(* IEC 61131-3 sources: programs/VI-54/VI-54_20171205/VI-54_20171205/Stations/PLC_VI54/VI-54_171014/Class/X_Axle_Correction, 1 file *)

(* ---- X_Axle_Correction.st ---- *)
(*!
<Class
	Name               = "X_Axle_Correction"
	Revision           = "0.0"
	RealtimeTask       = "false"
	CyclicTask         = "false"
	BackgroundTask     = "false"
	Sigmatek           = "false"
	OSInterface        = "false"
	HighPriority       = "false"
	Automatic          = "false"
	UpdateMode         = "Prescan"
	SharedCommandTable = "true"
	Objectsize         = "(750,120)">
	<Channels>
		<Server Name="CorrectionMM" Visualized="true" Initialize="false" WriteProtected="true" Retentive="false"/>
		<Server Name="StationNbr" Visualized="true" Initialize="false" WriteProtected="true" Retentive="false"/>
		<Server Name="X_Axle_Error" Visualized="true" Initialize="false" WriteProtected="true" Retentive="false"/>
		<Server Name="X_Axle_State" Visualized="true" Initialize="false" WriteProtected="true" Retentive="false"/>
		<Client Name="Comm_Next" Required="false" Internal="false"/>
		<Client Name="iFc_Trigger" Required="true" Internal="false"/>
		<Client Name="Standard3" Required="true" Internal="true"/>
		<Client Name="Virtual_Axle" Required="true" Internal="false"/>
		<Client Name="X_Axle" Required="true" Internal="false"/>
	</Channels>
	<Separators>
		<Servers>
			<SepChn Position="4"/>
			<SepChn Position="0"/>
		</Servers>
	</Separators>
	<Network Name="X_Axle_Correction">
		<!-- List of Components in this network -->
		<Components>
			<Object
				Name       = "_base"
				Class      = "MachineBase"
				Position   = "(324,120)"
				Visualized = "true">
				<Channels>
					<Server Name="ObjectServer"/>
					<Server Name="RunningMode"/>
					<Server Name="Stepper"/>
				</Channels>
			</Object>
			<Object
				Name           = "Standard3"
				Class          = "Standard"
				Position       = "(270,420)"
				Visualized     = "false"
				BackgroundTime = "1000 ms">
				<Channels>
					<Server Name="ClassSvr"/>
				</Channels>
			</Object>
		</Components>
		<Comments>
		</Comments>
		<!-- List of Connections in this network -->
		<Connections>
			<Connection Source="this.Standard3" Destination="Standard3.ClassSvr"/>
			<Connection Source="this.ObjectServer" Destination="_base.ObjectServer" Vertices="(1112,210),(940,210),"/>
			<Connection Source="this.Stepper" Destination="_base.Stepper" Vertices="(1112,270),(940,270),"/>
			<Connection Source="this.RunningMode" Destination="_base.RunningMode" Vertices="(1112,330),(940,330),"/>
		</Connections>
		<!-- Headerfiles -->
		<Options>
		</Options>
	</Network>
</Class>
*)
#pragma using MachineBase

X_Axle_Correction : CLASS
: MachineBase
  //Servers:
	StationNbr 	: SvrCh_DINT;
	X_Axle_State 	: SvrCh__LMCAXIS_STATUS;
	X_Axle_Error 	: SvrCh__LMCAXIS_ERROR;
	CorrectionMM 	: SvrCh_DINT;
  //Clients:
	iFc_Trigger 	: CltChCmd_ProductTriggerCamera;
	Virtual_Axle 	: CltChCmd__LMCAxis;
	X_Axle 	: CltChCmd__LMCAxis;
	Comm_Next 	: CltChCmd_X_Axle_Correction;
	Standard3 	: CltChCmd_Standard;
  //Variables:
		CalcAccDec 	: DINT;
		CalcSpeed 	: DINT;
		CameraPtr 	: ^StrCameraData;
		CalcLineSpeed 	: DINT;
		OldCleaningMode 	: OptiesEnum;
		CleaningSpeedOld 	: DINT;
		CalcCleaningSpeed 	: DINT;
		CalcCleaningAccDec 	: DINT;
		CleaningJogDistance 	: DINT;
		OldCalcLineSpeed 	: DINT;
		TriggerInfo 	: ProductTriggerCamera::OutInfoStr;
  //Functions:

	FUNCTION VIRTUAL GLOBAL MyInit;

	FUNCTION VIRTUAL GLOBAL MyCyTask;

	FUNCTION GLOBAL SetStationNbr
		VAR_INPUT
			Nbr 	: DINT;
		END_VAR;

	FUNCTION GLOBAL ChangePos
		VAR_INPUT
			Position 	: DINT;
		END_VAR;
  //Tables:
	FUNCTION @STD
		VAR_OUTPUT
			ret_code	: CONFSTATES;
		END_VAR;
	FUNCTION GLOBAL TAB @CT_;
END_CLASS;

#pragma using Standard
#pragma usingLtd _LMCAxis
#pragma usingLtd ProductTriggerCamera

FUNCTION GLOBAL X_Axle_Correction::MyInit

  // Set another inits
  if IsClientConnected(#Comm_Next) then
    Comm_Next.InitTask(SetGlobalPtr:= GlobalDataPtr, SetRecipePtr:= RecipePtr);
  end_if;

END_FUNCTION

FUNCTION GLOBAL X_Axle_Correction::MyCyTask

  // Set another CyTasks
  if IsClientConnected(#Comm_Next) then
    Comm_Next.CyTask();
  end_if;

  // Read Axle States
  X_Axle_State       := X_Axle.ReadAxisStatus();
  X_Axle_Error       := X_Axle.ReadAxisError();

  // Calculations
  CalcSpeed          := to_dint(to_real RecipePtr^.X_Axle.Speed ToMMperSec);
  CalcAccDec         := to_dint(to_real RecipePtr^.X_Axle.AccDec ToMMperSec);

  // Set Trigger info
  TriggerInfo        := iFc_Trigger.OffsetTrigger();

  // check for errors
  if GlobalDataPtr^.gGeneralData.NoError = 0 | GlobalDataPtr^.gGeneralData.iNoodstopOk = 0
    | GlobalDataPtr^.gRunStatus.gRunStatusGlob = eNoodstopStatus | GlobalDataPtr^.gRunStatus.gRunStatusGlob = eErrorStatus then
    if Stepper < 100 | Stepper >= 200 then
      Stepper := 100;
    end_if;
  end_if;

  case Stepper of
  00:// start
    if GlobalDataPtr^.gRunStatus.gRunStatusGlob = eRunStatus | GlobalDataPtr^.gRunStatus.gRunStatusGlob = eStartUpStatus
      | GlobalDataPtr^.gRunStatus.gRunStatusGlob = eCleaningStatus | GlobalDataPtr^.gRunStatus.gRunStatusGlob = ePauseStatus then
      if GlobalDataPtr^.gGeneralData.iDrivesOK = 1 then
        Stepper += 1;
      end_if;
    end_if;

  01:
    if GlobalDataPtr^.gGeneralData.iDrivesEnabled = 0 then  // Axles enabled??
      if X_Axle_State.PowerOn = 0 then
        X_Axle.PowerOn(Mode:= LMCAXIS_MOVE_ANY_WAY);
      end_if;
    else
      Stepper += 1;
    end_if;

  02: // What do we choose?
    GlobalDataPtr^.gRunStatus.gRunStatusXaxles[StationNbr] := GlobalDataPtr^.gRunStatus.gRunStatusGlob;
    if GlobalDataPtr^.gRunStatus.gRunStatusGlob = eStartUpStatus | GlobalDataPtr^.gRunStatus.gRunStatusGlob = eRunStatus
      | GlobalDataPtr^.gRunStatus.gRunStatusGlob = ePauseStatus then
      Stepper := 20;
    elsif GlobalDataPtr^.gRunStatus.gRunStatusGlob = eCleaningStatus then
      Stepper := 200;
    end_if;

  //--------------------------------
  20: // Reset positions of Axle
    X_Axle.SetPosition(Mode:=::_LMCAXIS_SETPOSITION::LMCAXIS_SET_ACTPOS_INTUNIT, Position:= 0);
    Stepper += 1;

  21: // Couple Axles to Virtual axle
    if X_Axle_State.DelayedMasterLock = false then
      X_Axle.CoupleGearAbsolute(MaxVel:= X_Axle.ReadParameter(ParNr:=::_LMCAXIS_READPARAMETER::LMCAXIS_PAR_RD_V_MAX, mode:= 0),
                                MaxAcc:= CalcAccDec,
                                DeltaPos:= 0,
                                pMaster:= Virtual_Axle.ReadMasterInfo(),
                                GearMul:= 1,
                                GearDiv:= 1);
    else
      Stepper += 1;
    end_if;

  22: // Check for runstatus
    GlobalDataPtr^.gRunStatus.gRunStatusXaxles[StationNbr] := GlobalDataPtr^.gRunStatus.gRunStatusGlob;
    if GlobalDataPtr^.gRunStatus.gRunStatusGlob = eStartUpStatus | GlobalDataPtr^.gRunStatus.gRunStatusGlob = eRunStatus
      | GlobalDataPtr^.gRunStatus.gRunStatusGlob = ePauseStatus then
      Stepper := 20;
    elsif GlobalDataPtr^.gRunStatus.gRunStatusGlob = eCleaningStatus then
      Stepper := 200;
    end_if;

  //--------------------------------
  40: // Set Line Speed
    GlobalDataPtr^.gRunStatus.gRunStatusXaxles[StationNbr] := eRunStatus;
    Virtual_Axle.MoveEndless(Speed:= CalcLineSpeed, Accel:= CalcAccDec);
    OldCalcLineSpeed := CalcLineSpeed;
    Stepper += 1;

  41: // Check for position difference
    if GlobalDataPtr^.gRunStatus.gRunStatusGlob <> eRunStatus & GlobalDataPtr^.gRunStatus.gRunStatusGlob <> ePauseStatus then
      Stepper := 100;
    elsif Standard3.R_TRIG(CLK:= TriggerInfo.TriggerState) = True then
      CorrectionMM += TriggerInfo.CameraData[StationNbr].Xposition;
      ChangePos(Position:= (CorrectionMM * 1000));
    elsif OldCalcLineSpeed <> CalcLineSpeed then
      Stepper -= 1;
    end_if;

  //--------------------------------
  100: // assen stopzetten en uitzetten
    GlobalDataPtr^.gRunStatus.gRunStatusXaxles[StationNbr] := eStopStatus;
    if X_Axle_State.PowerOn = 1 then
      X_Axle.PowerOff(Mode:= LMCAXIS_IMMEDIATE_STOPP);
    else
      Stepper += 1;
    end_if;

  101:
    GlobalDataPtr^.gRunStatus.gRunStatusXaxles[StationNbr] := eDriveOffStatus;
    if GlobalDataPtr^.gGeneralData.NoError = 1 & GlobalDataPtr^.gGeneralData.iNoodstopOk = 1 then
      Stepper := 0;
    end_if;

  //--------------------------------
  200: // Cleaning
    GlobalDataPtr^.gRunStatus.gRunStatusXaxles[StationNbr] := eCleaningStatus;
    OldCleaningMode := GlobalDataPtr^.gGeneralData.CleaningJogOption;
    if GlobalDataPtr^.gGeneralData.CleaningJogOption = Actief then
      Stepper := 205;
    else
      Stepper += 1;
    end_if;

  201: // Cleaning endless //
    X_Axle.MoveEndless(Speed:= CalcCleaningSpeed, Accel:= CalcCleaningAccDec);
    CleaningSpeedOld   := CalcCleaningSpeed;
    Stepper += 1;

  202:
    if GlobalDataPtr^.gRunStatus.gRunStatusGlob <> eCleaningStatus then
      Stepper := 100;
    elsif OldCleaningMode <> GlobalDataPtr^.gGeneralData.CleaningJogOption then // Is cleaningOption different?
      X_Axle.StopMove(Decel:= CalcCleaningAccDec);
      Stepper := 200;
    elsif CalcCleaningSpeed <> CleaningSpeedOld then
      Stepper -= 1;
    end_if;

  205: // Cleaning in jogmode (every time a step) //
    if GlobalDataPtr^.gRunStatus.gRunStatusGlob <> eCleaningStatus then
      Stepper := 100;
    elsif OldCleaningMode <> GlobalDataPtr^.gGeneralData.CleaningJogOption then // Is cleaningOption different?
      X_Axle.StopMove(Decel:= CalcCleaningAccDec);
      Stepper := 200;
    elsif GlobalDataPtr^.gGeneralData.CleaningJog = 1 then
      X_Axle.MoveRelative(Position:= CleaningJogDistance,
                          Mode:= LMCAXIS_MOVE_RELATIVE_TO_POSITION,
                          Speed:= CalcCleaningSpeed,
                          Accel:= CalcCleaningAccDec,
                          Decel:= CalcCleaningAccDec);
      Stepper += 1;
    end_if;

   206:
    if GlobalDataPtr^.gRunStatus.gRunStatusGlob <> eCleaningStatus then
      Stepper := 100;
    elsif X_Axle.InPosition(Mode:= LMCAXIS_SETPOS_IN_WINDOW_APP_UNITS, PositionWindow:= 1000) then
      if GlobalDataPtr^.gGeneralData.CleaningJog = 0 then
        Stepper -= 1;
      end_if;
    end_if;

  end_case;

END_FUNCTION

FUNCTION GLOBAL X_Axle_Correction::SetStationNbr
	VAR_INPUT
		Nbr 	: DINT;
	END_VAR

  StationNbr := Nbr;

  // Set station nbr
  if IsClientConnected(#Comm_Next) then
    Comm_Next.SetStationNbr(Nbr:= StationNbr + 1);
  end_if;

END_FUNCTION

FUNCTION GLOBAL X_Axle_Correction::ChangePos
	VAR_INPUT
		Position 	: DINT;
	END_VAR

  X_Axle.ChangeCoupleSettings(MaxVel:= X_Axle.ReadParameter(ParNr:=::_LMCAXIS_READPARAMETER::LMCAXIS_PAR_RD_V_MAX, mode:= 0),
                              MaxAcc:= CalcAccDec,
                              DeltaPos:= Position,
                              GearMul:= 1,
                              GearDiv:= 1);

END_FUNCTION
